PROGRAM MAIN
VAR
	bar : FooBar;
END_VAR

bar := FooBar.FOO_BAR_FIRST_VALUE;

END_PROGRAM

(* stored: Version 1.1.0.1, ProductVersion 3.1.4024.12
   POU MAIN: Id {69a6140f-d34b-4052-a7f3-57d0088fead9}, SpecialFunc None *)
